TYPE CyltronicProcessDataOut :
UNION
	CyltronicDataOutAct  : CyltronicProcessDataOutActual;
	CyltronicDataOutByte : CyltronicProcessDataOutBytes;
END_UNION
END_TYPE

(* stored: Version 1.1.0.1, ProductVersion 3.1.4024.10
   DUT CyltronicProcessDataOut: Id {cbc71a57-e834-46aa-a73a-ec7cf698a25f} *)
